FUNCTION And2 : BoolValue
VAR_INPUT
	value1 : BoolValue;
	value2 : BoolValue;
END_VAR
VAR
	p : POINTER TO BooleanExpression;
END_VAR

p := __NEW(BooleanExpression);

p^.Op2(
	operator := BooleanOperator.ANDop,
	value1 := value1,
	value2 := value2
);

And2 := p^;

END_FUNCTION

(* stored: Version 1.1.0.1
   POU And2: Id {6d1dbd7f-02dc-4cc7-804a-4a95b37f3620}, SpecialFunc None *)
